// Temperature monitor setpoints
{attribute 'qualified_only'}
VAR_GLOBAL PERSISTENT
    {attribute 'pytmc' := 'pv: @(BASE):LPS:TEMPMON01'}
    stTempMonSP01 : ST_TemperatureMonitorSetpoints;
    {attribute 'pytmc' := 'pv: @(BASE):LPS:TEMPMON02'}
    stTempMonSP02 : ST_TemperatureMonitorSetpoints;
    {attribute 'pytmc' := 'pv: @(BASE):LPS:TEMPMON03'}
    stTempMonSP03 : ST_TemperatureMonitorSetpoints;
    {attribute 'pytmc' := 'pv: @(BASE):LPS:TEMPMON04'}
    stTempMonSP04 : ST_TemperatureMonitorSetpoints;
    {attribute 'pytmc' := 'pv: @(BASE):LPS:TEMPMON05'}
    stTempMonSP05 : ST_TemperatureMonitorSetpoints;
    {attribute 'pytmc' := 'pv: @(BASE):LPS:TEMPMON06'}
    stTempMonSP06 : ST_TemperatureMonitorSetpoints;
    {attribute 'pytmc' := 'pv: @(BASE):LPS:TEMPMON07'}
    stTempMonSP07 : ST_TemperatureMonitorSetpoints;
    {attribute 'pytmc' := 'pv: @(BASE):LPS:TEMPMON08'}
    stTempMonSP08 : ST_TemperatureMonitorSetpoints;
END_VAR

(* stored: Version 1.1.0.1, ProductVersion 3.1.4022.18
   GVL GVL_TemperatureMonitor: Id {e923988d-0374-4c64-b59e-91da63738dbe} *)
